DATA_BLOCK "DB1_SYS"
TITLE = Datos de sistema
{ S7_Optimized_Access := 'TRUE' }
AUTHOR : ABH
VERSION : 0.1
NON_RETAIN
   VAR
      ON : Bool;   // Siempre a 1
      OFF : Bool;   // Siempre a 0
      SIM : Bool;   // Sistema en simulacion
      ACK : Bool;   // Acuse general de errores
      ARRANQUE : Bool;   // Marca de primer arranque del sistema
      Pulso100ms : Bool;   // Pulso 100 ms
      Pulso1seg : Bool;   // Pulso 1 segundo
      Pulso2seg : Bool;   // Pulso 2 segundo
      Pulso5seg : Bool;   // Pulso 5 segundos
      Pulso1min : Bool;   // Pulso 1 minuto
      Pulso1h : Bool;   // Pulso 1 hora
      FlipFlop1seg : Bool;   // Flip flop 1 seg ON - 1 seg OFF
      FlipFlop2seg : Bool;   // Flip flop 2 seg ON - 2 seg OFF
      FlipFlop5seg : Bool;   // Flip flop 5 seg ON - 5 seg OFF
      ResetEntidades { ExternalAccessible := 'False'; ExternalVisible := 'False'; ExternalWritable := 'False'} : Bool;   // Reset todas las entidades
      Reserva_18 : Bool;
      Pulsador : Struct
         EscribirFechaHora { S7_SetPoint := 'False'} : "UDT_ZC_PULSADOR";   // Pulsador cambio de fecha y hora desde hmi
         Ack { S7_SetPoint := 'False'} : Array[0..9] of "UDT_ZC_PULSADOR";   // Pulsador acuse general de errores
      END_STRUCT;
      FechaHoraActual {InstructionName := 'DTL'; LibVersion := '1.0'} : DTL;   // Fecha y hora actual del sistema
   END_VAR
   VAR RETAIN
      FechaHoraNueva {InstructionName := 'DTL'; LibVersion := '1.0'} : DTL;   // Fecha y hora nueva
   END_VAR
   VAR
      TiempoCiclo : Real;   // Tiempo de ciclo del PLC
   END_VAR
   VAR RETAIN
      Usuario : Struct
         Seleccion : Array[0..9] of Struct
            Orden : Bool;
            Usuario : String[25];
         END_STRUCT;
         Actual : String[25];   // Usuario actual
      END_STRUCT;
      Idioma : Struct
         Seleccionado : Int;   // Idioma seleccionado
         Espanol : Bool;   // Español
         Ingles : Bool;   // Ingles
         Aleman : Bool;   // Aleman
         Frances : Bool;   // Frances
         Portugues : Bool;   // Portugues
         Idioma_6 : Bool;
         Idioma_7 : Bool;
         Idioma_8 : Bool;
      END_STRUCT;
      Aux : Struct
         P_Trig_Pulso100ms : Bool;   // P_TRIG Pulso 100 ms
         P_Trig_Pulso1Seg : Bool;   // P_TRIG Pulso 1 segundo
         Contador2seg : USInt;   // Aux. Contador 2 segundos
         Contador5seg : USInt;   // Aux. Contador 5 segundos
         Contador1min : USInt;   // Aux. Contador 1 minuto
         Contador1h : UInt;   // Aux. Contador 1 hora
         auxRuntime : LReal;   // Aux. Runtime
      END_STRUCT;
   END_VAR


BEGIN
   ON := TRUE;
   OFF := FALSE;
   SIM := FALSE;
   ACK := FALSE;
   ARRANQUE := FALSE;
   Pulso100ms := FALSE;
   Pulso1seg := FALSE;
   Pulso2seg := FALSE;
   Pulso5seg := FALSE;
   Pulso1min := FALSE;
   Pulso1h := FALSE;
   FlipFlop1seg := TRUE;
   FlipFlop2seg := TRUE;
   FlipFlop5seg := TRUE;
   ResetEntidades := FALSE;
   Reserva_18 := FALSE;
   Pulsador.EscribirFechaHora.Hmi := FALSE;
   Pulsador.EscribirFechaHora.Plc := FALSE;
   Pulsador.EscribirFechaHora.Permiso := TRUE;
   Pulsador.EscribirFechaHora.Visibilidad := TRUE;
   Pulsador.EscribirFechaHora.AuxPulso := FALSE;
   Pulsador.EscribirFechaHora.AuxTiempo := 0;
   Pulsador.Ack[0].Hmi := FALSE;
   Pulsador.Ack[0].Plc := FALSE;
   Pulsador.Ack[0].Permiso := TRUE;
   Pulsador.Ack[0].Visibilidad := FALSE;
   Pulsador.Ack[0].AuxPulso := FALSE;
   Pulsador.Ack[0].AuxTiempo := 0;
   Pulsador.Ack[1].Hmi := FALSE;
   Pulsador.Ack[1].Plc := FALSE;
   Pulsador.Ack[1].Permiso := TRUE;
   Pulsador.Ack[1].Visibilidad := FALSE;
   Pulsador.Ack[1].AuxPulso := FALSE;
   Pulsador.Ack[1].AuxTiempo := 0;
   Pulsador.Ack[2].Hmi := FALSE;
   Pulsador.Ack[2].Plc := FALSE;
   Pulsador.Ack[2].Permiso := TRUE;
   Pulsador.Ack[2].Visibilidad := FALSE;
   Pulsador.Ack[2].AuxPulso := FALSE;
   Pulsador.Ack[2].AuxTiempo := 0;
   Pulsador.Ack[3].Hmi := FALSE;
   Pulsador.Ack[3].Plc := FALSE;
   Pulsador.Ack[3].Permiso := TRUE;
   Pulsador.Ack[3].Visibilidad := FALSE;
   Pulsador.Ack[3].AuxPulso := FALSE;
   Pulsador.Ack[3].AuxTiempo := 0;
   Pulsador.Ack[4].Hmi := FALSE;
   Pulsador.Ack[4].Plc := FALSE;
   Pulsador.Ack[4].Permiso := TRUE;
   Pulsador.Ack[4].Visibilidad := FALSE;
   Pulsador.Ack[4].AuxPulso := FALSE;
   Pulsador.Ack[4].AuxTiempo := 0;
   Pulsador.Ack[5].Hmi := FALSE;
   Pulsador.Ack[5].Plc := FALSE;
   Pulsador.Ack[5].Permiso := TRUE;
   Pulsador.Ack[5].Visibilidad := FALSE;
   Pulsador.Ack[5].AuxPulso := FALSE;
   Pulsador.Ack[5].AuxTiempo := 0;
   Pulsador.Ack[6].Hmi := FALSE;
   Pulsador.Ack[6].Plc := FALSE;
   Pulsador.Ack[6].Permiso := TRUE;
   Pulsador.Ack[6].Visibilidad := FALSE;
   Pulsador.Ack[6].AuxPulso := FALSE;
   Pulsador.Ack[6].AuxTiempo := 0;
   Pulsador.Ack[7].Hmi := FALSE;
   Pulsador.Ack[7].Plc := FALSE;
   Pulsador.Ack[7].Permiso := TRUE;
   Pulsador.Ack[7].Visibilidad := FALSE;
   Pulsador.Ack[7].AuxPulso := FALSE;
   Pulsador.Ack[7].AuxTiempo := 0;
   Pulsador.Ack[8].Hmi := FALSE;
   Pulsador.Ack[8].Plc := FALSE;
   Pulsador.Ack[8].Permiso := TRUE;
   Pulsador.Ack[8].Visibilidad := FALSE;
   Pulsador.Ack[8].AuxPulso := FALSE;
   Pulsador.Ack[8].AuxTiempo := 0;
   Pulsador.Ack[9].Hmi := FALSE;
   Pulsador.Ack[9].Plc := FALSE;
   Pulsador.Ack[9].Permiso := TRUE;
   Pulsador.Ack[9].Visibilidad := FALSE;
   Pulsador.Ack[9].AuxPulso := FALSE;
   Pulsador.Ack[9].AuxTiempo := 0;
   FechaHoraActual.YEAR := 2025;
   FechaHoraActual.MONTH := 9;
   FechaHoraActual.DAY := 18;
   FechaHoraActual.WEEKDAY := 5;
   FechaHoraActual.HOUR := 19;
   FechaHoraActual.MINUTE := 1;
   FechaHoraActual.SECOND := 56;
   FechaHoraActual.NANOSECOND := 550304800;
   FechaHoraActual := DTL#2025-09-18-19:01:56.550304800;
   FechaHoraNueva.YEAR := 2024;
   FechaHoraNueva.MONTH := 8;
   FechaHoraNueva.DAY := 19;
   FechaHoraNueva.WEEKDAY := 2;
   FechaHoraNueva.HOUR := 12;
   FechaHoraNueva.MINUTE := 12;
   FechaHoraNueva.SECOND := 12;
   FechaHoraNueva.NANOSECOND := 215955351;
   FechaHoraNueva := DTL#2024-08-19-12:12:12.215955351;
   TiempoCiclo := 28.34702;
   Usuario.Seleccion[0].Orden := FALSE;
   Usuario.Seleccion[0].Usuario := 'sive';
   Usuario.Seleccion[1].Orden := FALSE;
   Usuario.Seleccion[1].Usuario := '';
   Usuario.Seleccion[2].Orden := FALSE;
   Usuario.Seleccion[2].Usuario := '';
   Usuario.Seleccion[3].Orden := FALSE;
   Usuario.Seleccion[3].Usuario := '';
   Usuario.Seleccion[4].Orden := FALSE;
   Usuario.Seleccion[4].Usuario := '';
   Usuario.Seleccion[5].Orden := FALSE;
   Usuario.Seleccion[5].Usuario := 's';
   Usuario.Seleccion[6].Orden := FALSE;
   Usuario.Seleccion[6].Usuario := '';
   Usuario.Seleccion[7].Orden := FALSE;
   Usuario.Seleccion[7].Usuario := '';
   Usuario.Seleccion[8].Orden := FALSE;
   Usuario.Seleccion[8].Usuario := '';
   Usuario.Seleccion[9].Orden := FALSE;
   Usuario.Seleccion[9].Usuario := '';
   Usuario.Actual := 's';
   Idioma.Seleccionado := 0;
   Idioma.Espanol := TRUE;
   Idioma.Ingles := FALSE;
   Idioma.Aleman := FALSE;
   Idioma.Frances := FALSE;
   Idioma.Portugues := FALSE;
   Idioma.Idioma_6 := FALSE;
   Idioma.Idioma_7 := FALSE;
   Idioma.Idioma_8 := FALSE;
   Aux.P_Trig_Pulso100ms := TRUE;
   Aux.P_Trig_Pulso1Seg := TRUE;
   Aux.Contador2seg := 0;
   Aux.Contador5seg := 0;
   Aux.Contador1min := 33;
   Aux.Contador1h := 573;
   Aux.auxRuntime := 3.12728340475131E-308;

END_DATA_BLOCK

